TYPE ServicesProcesses :
STRUCT
	///Start initializing
	initialize: Process;
	///Lock the system
	lock: Process;
	///Unlock the system
	unlock: Process;
	///Change the operating state (e.g. AUTO, MANUAL, ...)
	changeOperatingState: ChangeOperatingStateProcess;
END_STRUCT
END_TYPE

(* stored: Version 1.1.0.1, ProductVersion 3.1.4019.2
   DUT ServicesProcesses: Id {a0fccae4-c47b-436c-bc70-2ee33033daa6} *)
